(*
SPDX-FileCopyrightText: © 2026 Oleksandr Tiutyk <trofimich@gmail.com>
SPDX-License-Identifier: MIT
License: https://opensource.org/license/mit
*)

(*!
<summary>Exposes compiler-initialized namespace storage to library objects.</summary>
<description>
The internal extractor supplies the namespace of this library. Returned references borrow program-owned
storage while the provider is live and must not be modified. Reacquire them after reinitialization or
relocation. No lazy initialization or allocation occurs.
</description>
*)

{attribute 'no_explicit_call' := 'do not call this function block directly'}
PROGRAM INTERNAL CurrentNamespace
VAR
	{attribute 'hide'} 
	_NamespaceExtractor : NamespaceExtractor;

	{attribute 'hide'}
	_ClassName : STRING := __POUNAME();
END_VAR

(*!
<summary>Borrows the library namespace string.</summary>
<description>
Storage belongs to the internal program. Callers must not mutate it or retain it across application unloading.
</description>
*)
{attribute 'monitoring' := 'call'}
PROPERTY Name : REFERENCE TO STRING
GET
Name REF= _NamespaceExtractor.CurrentNamespace;
END_GET
END_PROPERTY

(*!
<summary>Borrows the diagnostic name of this internal program.</summary>
<description>
Returns program-owned read-only storage; does not initialize or allocate another object.
</description>
*)
{attribute 'monitoring' := 'call'}
PROPERTY ClassName : REFERENCE TO STRING
GET
ClassName REF= _ClassName;
END_GET
END_PROPERTY

(*!
<summary>Borrows the compiler-initialized namespace of this library.</summary>
<description>
Returns the same storage as Name without recursion or ownership transfer.
</description>
*)
{attribute 'monitoring' := 'call'}
PROPERTY NamespaceName : REFERENCE TO STRING
GET
NamespaceName REF= _NamespaceExtractor.CurrentNamespace;
END_GET
END_PROPERTY

END_PROGRAM

(* stored: Version 1.1.0.1
   POU CurrentNamespace: Id {3d358878-e58a-48fc-b41d-ea218a9e3a9b}, SpecialFunc None
   Property Name: Id {7cbbb419-2ca8-4daf-a0f2-920d8419554e}
   Get Get: Id {50d77bfb-1d4f-44a3-b3a6-73039375ff9c}
   Property ClassName: Id {2ebd4d8d-68eb-4b0a-bcb4-ec3e1a8d2258}
   Get Get: Id {bdc41251-97be-4ace-ac04-b0895b8868ac}
   Property NamespaceName: Id {f68b9c38-865d-4cff-97ec-b1dccffff72b}
   Get Get: Id {20a98e82-9c34-46f2-8ac9-0eae5731c9d6} *)
